Staubli VAL3: insertItem.pgx

public program insertItem(num& x_nIndexCopy, num x_nIndexPaste)
  local num l_nLastType
  local point l_pPoint
  local num l_nType
begin
  //
  // use to add more elements from the typical one
  //
  // insert all the field
  //
  l_pPoint=pEditPoint.tData[x_nIndexCopy].pPoint
  link(pEditPoint.tData[x_nIndexPaste].pPoint,pEditPoint.fFrame)
  insert(pEditPoint.tData[x_nIndexPaste])
  // set IT
  pEditPoint.tData[x_nIndexPaste].pPoint.trsf=l_pPoint.trsf
end
